FUNCTION_BLOCK FB_EL6001_LINE_CTRL
VAR_IN_OUT
	EL6001 : TYP_HW_EL6001;

END_VAR
VAR_INPUT
END_VAR
VAR_OUTPUT
END_VAR
VAR
	SerialLineControl : SerialLineControl;
	Buffer : TYP_SERIAL_DATA;
END_VAR

SerialLineControl.Mode := ComSerialLineMode_t.SERIALLINEMODE_EL6_22B;
SerialLineControl.pComIn := ADR(EL6001.In.COM);
SerialLineControl.pComOut := ADR(EL6001.Out.COM);
SerialLineControl.SizeComIn := UINT_TO_INT(SIZEOF(EL6001.In.COM));
SerialLineControl(RxBuffer := Buffer.RxData, TxBuffer := Buffer.TxData);

PROPERTY PUBLIC RxBuffer : REFERENCE TO COMbuffer
GET
RxBuffer REF= THIS^.Buffer.RxData;
END_GET
END_PROPERTY

PROPERTY PUBLIC TxBuffer : REFERENCE TO COMbuffer
GET
TxBuffer REF= THIS^.Buffer.TxData;
END_GET
END_PROPERTY

END_FUNCTION_BLOCK

(* stored: Version 1.1.0.1, ProductVersion 3.1.4024.12
   POU FB_EL6001_LINE_CTRL: Id {df7462e1-ad58-4b3e-bdae-a9ae649e5322}, SpecialFunc None
   Property RxBuffer: Id {4b2e2131-5397-484a-99cc-f0bca36fa536}
   Get Get: Id {04f4a679-9ff6-402c-840c-d3416344bc22}
   Property TxBuffer: Id {85ebcbad-5070-451a-8656-dcd393a6893f}
   Get Get: Id {3a754f51-453e-4e1c-a9b4-e9bca9a59081} *)
